(* IEC 61131-3 sources: factoryforge/examples/openplc/roller-line-weighing, 1 file *)

(* ---- roller_line_weighing.st ---- *)
(* ------------------------------------------------------------------------
   FactoryForge starter -- Roller line with weighing (scene roller-line-weighing)
   OpenPLC Runtime v3, IEC 61131-3 Structured Text, over Modbus TCP.
   Generated by tools/gen_starters.py from the scene's tag set; see README.md
   beside this file. Write your program in section 2 below.

   THE TASK
     Checkweigh. Judge each carton on the peak weight it shows as it
     crosses the deck, and reject anything over the limit on the panel's
     pot. The inductive sensor sees metal only, and on this line the steel
     cartons are also the heavy ones -- so two independent instruments
     should agree.

   DONE WHEN
     The cartons you flag over-limit are the same ones the inductive sensor
     flags as metal. Watch the spacing: two cartons on the deck at once
     read as one peak, so a real checkweigher line holds the feed while the
     scale is loaded.

   HOW IT IS WIRED
     FactoryForge is the Modbus slave; OpenPLC is the master and polls it.
     mbconfig.cfg beside this file is that Slave Device. The addresses
     below are the ones the sidecar serves for this scene when it is
     started AFTER the scene is open:

       factoryforge-sidecar connect --driver modbus-tcp -o port 5502

     It prints its address map on startup; that map is the authority, and
     the table below must match it line for line. Change scene and the
     sidecar keeps every address it has handed out and puts new tags above
     them -- restart it after changing scene.

     OpenPLC numbers each block it polls from 100: slave coil n is
     %QX(100 + n/8).(n mod 8), slave input register n is %IW(100 + n).

     An INT or REAL tag is 32 bits and takes TWO registers, high word
     first. Section 1 rebuilds the inputs and section 3 splits the outputs;
     your program works with the plain DINT and REAL variables.

     In the sidecar's order (block, then address; addresses are decimal):

     MODBUS   REGS  OPENPLC                TAG
     0x0      1     %QX100.0               emitter.emit
     0x1      1     %QX100.1               infeed.rotate
     0x2      1     %QX100.2               panel.green
     0x3      1     %QX100.3               panel.red
     0x4      1     %QX100.4               scale.rotate
     1x0      1     %IX100.0               infeed.fault
     1x1      1     %IX100.1               metal_check.detect
     1x2      1     %IX100.2               panel.estop
     1x3      1     %IX100.3               panel.reset
     1x4      1     %IX100.4               panel.start
     1x5      1     %IX100.5               panel.stop
     1x6      1     %IX100.6               scale.fault
     4x0      2     %QW100 + %QW101        weight_readout.value
     3x0      2     %IW100 + %IW101        outfeed.count
     3x2      2     %IW102 + %IW103        panel.setpoint
     3x4      2     %IW104 + %IW105        scale.weight
   ------------------------------------------------------------------------ *)

(* The sidecar sends a 32-bit value as two registers, high word first
   (struct.pack(">i") in drivers/modbus_tcp.py). DWORD_TO_DINT reinterprets
   the bit pattern, so this is right for negative values too. *)
FUNCTION FF_WORDS_TO_DINT : DINT
  VAR_INPUT
    HI : WORD;
    LO : WORD;
  END_VAR
  FF_WORDS_TO_DINT := DWORD_TO_DINT(SHL(IN := WORD_TO_DWORD(HI), N := 16)
                                    OR WORD_TO_DWORD(LO));
END_FUNCTION

(* A REAL arrives the same way: IEEE-754 single precision, high word first.
   OpenPLC's DWORD_TO_REAL cannot rebuild it -- it converts the NUMBER, so
   16#3F800000 becomes 1065353216.0 rather than 1.0 -- so this takes the
   sign, exponent and mantissa apart by hand. Exact for every normal value;
   zero and the tiny subnormals (below 1.2E-38) come back as 0.0. *)
FUNCTION FF_WORDS_TO_REAL : REAL
  VAR_INPUT
    HI : WORD;
    LO : WORD;
  END_VAR
  VAR
    Exponent : INT;
    Value    : REAL;
  END_VAR
  Exponent := WORD_TO_INT(SHR(IN := HI, N := 7) AND 16#00FF);
  IF Exponent = 0 OR Exponent = 255 THEN
    Value := 0.0;
  ELSE
    Value := 1.0 + DWORD_TO_REAL(SHL(IN := WORD_TO_DWORD(HI AND 16#007F), N := 16)
                                 OR WORD_TO_DWORD(LO)) / 8388608.0;
    Exponent := Exponent - 127;
    WHILE Exponent > 0 DO
      Value := Value * 2.0;
      Exponent := Exponent - 1;
    END_WHILE;
    WHILE Exponent < 0 DO
      Value := Value / 2.0;
      Exponent := Exponent + 1;
    END_WHILE;
    IF (HI AND 16#8000) <> 0 THEN
      Value := -Value;
    END_IF;
  END_IF;
  FF_WORDS_TO_REAL := Value;
END_FUNCTION

PROGRAM roller_line_weighing
  VAR
    (* --- PLC writes: coils --------------------------------------------- *)
    EmitterEmit  AT %QX100.0  : BOOL;  (* emitter.emit  0x0   rising edge = feed one carton; hold each level well over one poll; every 3rd carton is steel *)
    InfeedRotate AT %QX100.1  : BOOL;  (* infeed.rotate 0x1   run the roller deck *)
    PanelGreen   AT %QX100.2  : BOOL;  (* panel.green   0x2   green lamp on the panel *)
    PanelRed     AT %QX100.3  : BOOL;  (* panel.red     0x3   red lamp on the panel *)
    ScaleRotate  AT %QX100.4  : BOOL;  (* scale.rotate  0x4   run the weighing belt *)
    (* --- PLC writes: holding registers, two per value ------------------ *)
    WeightReadoutValueHi AT %QW100    : WORD;  (* weight_readout.value 4x0   high word of WeightReadoutValue *)
    WeightReadoutValueLo AT %QW101    : WORD;  (* weight_readout.value 4x1   low word of WeightReadoutValue *)
    (* --- PLC reads: discrete inputs ------------------------------------ *)
    InfeedFault      AT %IX100.0  : BOOL;  (* infeed.fault       1x0   drive fault: TRUE = faulted; a faulted drive does not turn *)
    MetalCheckDetect AT %IX100.1  : BOOL;  (* metal_check.detect 1x1   TRUE while a METAL carton is in front of it; cardboard is invisible to it *)
    PanelEstop       AT %IX100.2  : BOOL;  (* panel.estop        1x2   E-stop, normally closed: TRUE = healthy, FALSE = pressed; stays pressed until pulled out *)
    PanelReset       AT %IX100.3  : BOOL;  (* panel.reset        1x3   Reset button, momentary: a short pulse per press *)
    PanelStart       AT %IX100.4  : BOOL;  (* panel.start        1x4   Start button, momentary: a short pulse per press -- latch it *)
    PanelStop        AT %IX100.5  : BOOL;  (* panel.stop         1x5   Stop button, momentary: a short pulse per press *)
    ScaleFault       AT %IX100.6  : BOOL;  (* scale.fault        1x6   drive fault: TRUE = faulted; a faulted drive does not turn *)
    (* --- PLC reads: input registers, two per value --------------------- *)
    OutfeedCountHi  AT %IW100    : WORD;  (* outfeed.count  3x0   high word of OutfeedCount *)
    OutfeedCountLo  AT %IW101    : WORD;  (* outfeed.count  3x1   low word of OutfeedCount *)
    PanelSetpointHi AT %IW102    : WORD;  (* panel.setpoint 3x2   high word of PanelSetpoint *)
    PanelSetpointLo AT %IW103    : WORD;  (* panel.setpoint 3x3   low word of PanelSetpoint *)
    ScaleWeightHi   AT %IW104    : WORD;  (* scale.weight   3x4   high word of ScaleWeight *)
    ScaleWeightLo   AT %IW105    : WORD;  (* scale.weight   3x5   low word of ScaleWeight *)
  END_VAR

  (* A second VAR block, and not for tidiness: matiec will not mix located
     and unlocated declarations in one. Your own variables go here too. *)
  VAR
    (* --- PLC reads, in engineering units ---------------------------------- *)
    OutfeedCount       : DINT;  (* outfeed.count  cartons this remover has taken off the line, running total *)
    PanelSetpoint      : REAL;  (* panel.setpoint the operator's pot, 0..6000 g (starts at 3000) *)
    ScaleWeight        : DINT;  (* scale.weight   load cell: grams on the deck right now (everything on it, not one carton) *)
    (* --- PLC writes, in engineering units ---------------------------------- *)
    WeightReadoutValue : DINT;  (* weight_readout.value number shown on the display (g) *)
    Raw32 : DWORD;  (* scratch for splitting a 32-bit output *)
  END_VAR

  (* ===== 1. Inputs: rebuild each 32-bit value from its two registers ===== *)
  OutfeedCount := FF_WORDS_TO_DINT(HI := OutfeedCountHi, LO := OutfeedCountLo);
  PanelSetpoint := FF_WORDS_TO_REAL(HI := PanelSetpointHi, LO := PanelSetpointLo);
  ScaleWeight := FF_WORDS_TO_DINT(HI := ScaleWeightHi, LO := ScaleWeightLo);

  (* ===== 2. Your program ================================================
     The task is at the top of this file and in the scene's Task panel.
     Every signal above can be used by name here: the bits directly, the
     32-bit values through OutfeedCount, PanelSetpoint, ScaleWeight,
     WeightReadoutValue. *)

  (* ===== 3. Outputs: split each 32-bit value into its two registers ===== *)
  Raw32 := DINT_TO_DWORD(WeightReadoutValue);
  WeightReadoutValueHi := DWORD_TO_WORD(SHR(IN := Raw32, N := 16));
  WeightReadoutValueLo := DWORD_TO_WORD(Raw32);

END_PROGRAM

CONFIGURATION Config0

  RESOURCE Res0 ON PLC
    (* 20 ms, as in examples/openplc/Sorting.st: every scan spent waiting
       comes out of the scene's timing margins. *)
    TASK Main(INTERVAL := T#20ms, PRIORITY := 0);
    PROGRAM Inst0 WITH Main : roller_line_weighing;
  END_RESOURCE

END_CONFIGURATION
